FUNCTION_BLOCK Part EXTENDS ITF_Cyclic
VAR_INPUT
END_VAR
VAR_OUTPUT
END_VAR
VAR
END_VAR

END_FUNCTION_BLOCK

(* stored: Version 1.1.0.1, ProductVersion 3.1.4024.12
   POU Part: Id {c6022a1a-ace8-47d1-b56d-00a06f3159aa}, SpecialFunc None *)
